(*
SPDX-FileCopyrightText: © 2026 Oleksandr Tiutyk <trofimich@gmail.com>
SPDX-License-Identifier: MIT
License: https://opensource.org/license/mit
*)

INTERFACE IArgumentOutOfRangeException EXTENDS IGeneralException

METHOD Throw
VAR_INPUT
	sourceNamespaceName : STRING;
	sourceClassName : STRING;
	sourcePOUName : STRING;
	sourcePosition : STRING;
	argumentName : STRING;
	argumentValue : ANY;
END_VAR
END_METHOD

END_INTERFACE

(* stored: Version 1.1.0.1
   Itf IArgumentOutOfRangeException: Id {b593408e-8234-4422-a350-6b47381deafa}
   Method Throw: Id {3a3b6fab-8c6a-43b0-a149-d2423f42faeb} *)
